{attribute 'GeneratedUsingTerminal: EL2032-0000-0018'}
{attribute addProperty BoxType "EL2032-0000-0018"}
{attribute addProperty Id "OutputAT %Q*BOOL1"}
{attribute addProperty CRC "1120571895"}
{attribute addProperty Size "1"}
TYPE Channel_42CA91F7 EXTENDS OutputBase_10CEE7DE :
STRUCT
	{attribute addProperty Name "Output"}
	Output AT %Q* : BOOL;
END_STRUCT
END_TYPE

(* stored: Version 1.2.0.0, ProductVersion 3.1.4024.9
   DUT Channel_42CA91F7: Id {ed4e67bf-0fa4-4131-893a-8481113013a4} *)
